PROGRAM MAIN
VAR
END_VAR

END_PROGRAM

(* stored: Version 1.1.0.1
   POU MAIN: Id {442695f4-4c33-4ebb-b326-988b190a2c4b} *)
